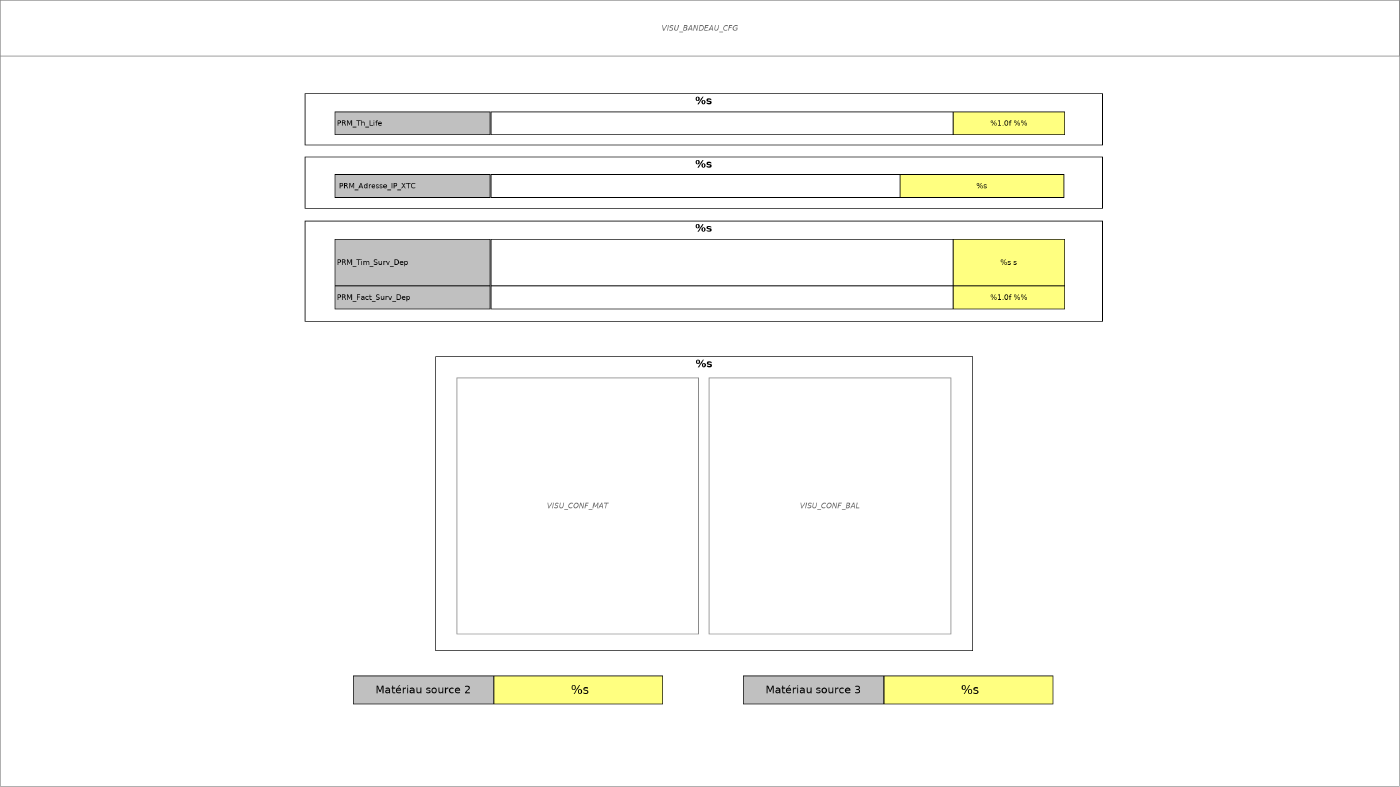
VISUALIZATION VISU_CONFIG_EVAP  // 1920x1080, background image fond_blanc_1280_1024
    Frame (0,0 1920x77)
        shows VISU_BANDEAU_CFG()
    RoundedRectangle (597,489 737x404), "%s", text list: 'TextList_Config_Evap', text index: 5
    RoundedRectangle (418,215 1094x71), "%s", text list: 'TextList_Config_Evap', text index: 20
    RoundedRectangle (418,128 1094x71), "%s", text list: 'TextList_Config_Evap', text index: 0
    Group (459,153 1001x32)
        Rectangle (214,0 634x32), text list: 'TextList_Config_Evap', text index: 1
        Rectangle (848,0 153x32), "%1.0f %%", text variable: PRG_EVAP.PRM_Seuil_Crystal_Life, input disabled if: NOT Global_Variables.PRG_USER.ACTU_USER.CONF_MACHINE
            OnMouseClick: write the text variable via InputWithLimits, min 0, max 100
        Rectangle (0,0 213x32), "PRM_Th_Life"
    RoundedRectangle (418,303 1094x138), "%s", text list: 'TextList_Config_Evap', text index: 2
    Rectangle (673,328 634x64), text list: 'TextList_Config_Evap', text index: 3
    Rectangle (1307,328 153x64), "%s s", text variable: PRG_EVAP.EVAPS1.PRM_TPS_MIN_SURV_DEPOT, input disabled if: NOT Global_Variables.PRG_USER.ACTU_USER.CONF_MACHINE
        OnMouseClick: write the text variable via InputWithLimits, min 0
    Rectangle (459,328 213x64), "PRM_Tim_Surv_Dep"
    Rectangle (673,392 634x32), text list: 'TextList_Config_Evap', text index: 4
    Rectangle (1307,392 153x32), "%1.0f %%", text variable: PRG_EVAP.EVAPS1.PRM_FACTEUR_TEMPS_DEPOT, input disabled if: NOT Global_Variables.PRG_USER.ACTU_USER.CONF_MACHINE
        OnMouseClick: write the text variable via InputWithLimits, min 0
    Rectangle (459,392 213x32), "PRM_Fact_Surv_Dep"
    Group (459,239 1000x32)
        Rectangle (0,0 213x32), "PRM_Adresse_IP_XTC", text variable: 1
        Rectangle (214,0 562x32), text list: 'TextList_Config_Evap', text index: 21
        Rectangle (775,0 225x32), "%s", text variable: Global_Variables.PRG_EVAP.PRM_Adresse_IP_XTC, input disabled if: NOT Global_Variables.PRG_USER.ACTU_USER.CONF_MACHINE
            OnMouseDown: write the text variable via InputWithLimits
    Frame (626,518 332x352)
        shows VISU_CONF_MAT(m_Input_CRUCIBLE := PRG_EVAP.CRUCIBLE1)
    Frame (972,518 332x352)
        shows VISU_CONF_BAL(m_Input_SWEEP := PRG_EVAP.SWEEP1)
    Rectangle (484,927 193x39), "Matériau source 2"
    Rectangle (677,927 232x39), "%s", text variable: Global_Variables.PRG_EVAP.PRM_Mat_Source2, input disabled if: NOT Global_Variables.PRG_USER.ACTU_USER.CONF_MACHINE
        OnMouseDown: write the text variable via InputWithLimits
    Rectangle (1019,927 193x39), "Matériau source 3"
    Rectangle (1212,927 232x39), "%s", text variable: Global_Variables.PRG_EVAP.PRM_Mat_Source3, input disabled if: NOT Global_Variables.PRG_USER.ACTU_USER.CONF_MACHINE
        OnMouseDown: write the text variable via InputWithLimits
END_VISUALIZATION

(* stored: Version 1.1.0.1, ProductVersion 3.1.4026.18
   Visu VISU_CONFIG_EVAP: Id {6a7a909a-ae23-42fe-8ed9-ebe43168096e} *)
